Omron Sysmac Studio project IoTSampleProjectNX1P2_9 (Sysmac Studio 1.47.0.64008, StandardProject)

# Controller new_Controller_0: NX1P2-9024DT1 version 1.47
Task PrimaryTask (priority 4, period or condition 2000): MQTT_AWS, DynamoDB_AWS
Library OmronLib_MQTT_Comm_V1_0 1.0.0 (contents left out)

PROGRAM MQTT_AWS
VAR
    trigger1 : BOOL;
    ClientID : STRING[256];
    ConnectionSettings : OmronLib\MQTT_Comm\sConnectionSettings;
    Pub_Topic : STRING[512];
    Pub_PubMsg : STRING[256];
    Pub_PubSettings : OmronLib\MQTT_Comm\sPubFlags;
    Sub_Topic : STRING[512];
    ClientReference : OmronLib\MQTT_Comm\sClientReference;
    KeepAlive : UINT;
    Timeout : UINT;
    DiscardMsgTime : UINT;
    busy : BOOL;
    DiscardMsgNum : UDINT;
    SessionPresent : BOOL;
    error : BOOL;
    errorid : WORD;
    erroridex : DWORD;
    MQTTClient00 : OmronLib\MQTT_Comm\MQTTClient;
    MQTTPubString : OmronLib\MQTT_Comm\MQTTPubString;
    Pub_PacketID : UINT;
    Pub_MsgType : USINT;
    Put_Timeout : UINT;
    pub_busy : BOOL;
    pub_error : BOOL;
    pub_errorid : WORD;
    pub_erroridex : DWORD;
    MQTT : OmronLib\MQTT_Comm\MQTTSubString;
    MQTTSubString00 : OmronLib\MQTT_Comm\MQTTSubString;
    MQTTPubString00 : OmronLib\MQTT_Comm\MQTTPubString;
    Sub_RcvMsg : STRING[1986];
    Sub_SubQos : BYTE;
    Sub_Timeout : UINT;
    Sub_Status : SINT;
    Sub_Received : BOOL;
    Sub_RcvTopic : STRING[512];
    sub_error : BOOL;
    sub_errorid : WORD;
    sub_erroridex : DWORD;
    trigger2 : BOOL;
    MQTTPing00 : OmronLib\MQTT_Comm\MQTTPing;
    ping_Timeout : UINT;
    ping_busy : BOOL;
    Ping_elapsedtime : UINT;
    ping_error : BOOL;
    ping_errorid : WORD;
    ping_erroridex : DWORD;
    trigger3 : BOOL;
    trigger4 : BOOL;
    Pub_Timeout : UINT;
    trigger5 : BOOL;
    MQTTPubAry00 : OmronLib\MQTT_Comm\MQTTPubAryByte;
    Pub_MsgAry : ARRAY[0..65534] OF BYTE;
    Pub_MsgSize : UINT;
    pubary_busy : BOOL;
    pubary_error : BOOL;
    pubary_errorid : WORD;
    pubary_erroridex : DWORD;
    trigger6 : BOOL;
    MQTTSubAry00 : OmronLib\MQTT_Comm\MQTTSubAryByte;
    SubAry_RcvMsg : ARRAY[0..65534] OF BYTE;
    SubAry_SubQoS : BYTE;
    Subary_Status : SINT;
    SubAry_Received : BOOL;
    SubAry_MsgSize : UINT;
    SubAry_RcvTopic : STRING[512];
    subary_error : BOOL;
    subary_errorid : WORD;
    subary_erroridex : DWORD;
    RcvMsg : STRING[1986];
    tmpAryStr : ARRAY[0..1985] OF BYTE;
END_VAR
VAR
    _e1 : R_TRIG;
    _e2 : R_TRIG;
    _e3 : R_TRIG;
END_VAR

(* Section Section0: ladder, written here as Structured Text *)

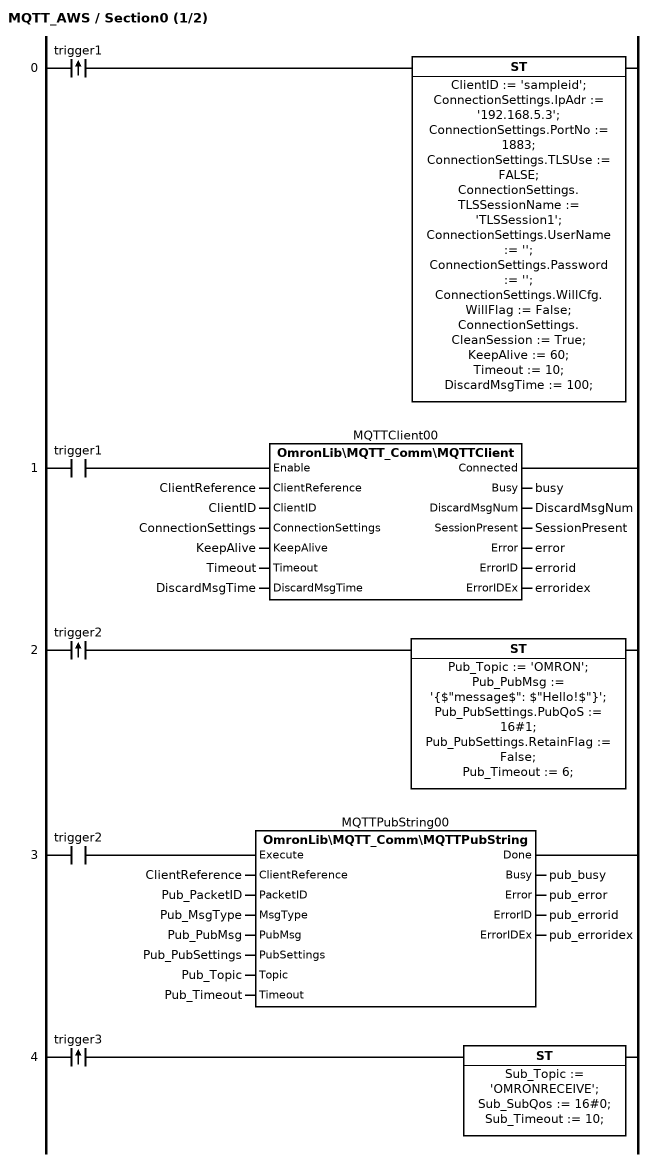
(* Rung 0 *)
_e1(CLK := trigger1);
IF _e1.Q THEN
    ClientID := 'sampleid';
    
    ConnectionSettings.IpAdr := '192.168.5.3';
    ConnectionSettings.PortNo := 1883;
    ConnectionSettings.TLSUse := FALSE;
    
    ConnectionSettings.TLSSessionName := 'TLSSession1';
    
    ConnectionSettings.UserName := '';
    ConnectionSettings.Password := '';
    ConnectionSettings.WillCfg.WillFlag := False;
    ConnectionSettings.CleanSession := True;
    
    KeepAlive := 60;
    Timeout := 10;
    DiscardMsgTime := 100;
END_IF;
(* Rung 1 *)
MQTTClient00(Enable := trigger1, ClientReference := ClientReference, ClientID := ClientID, ConnectionSettings := ConnectionSettings, KeepAlive := KeepAlive, Timeout := Timeout, DiscardMsgTime := DiscardMsgTime, Busy => busy, DiscardMsgNum => DiscardMsgNum, SessionPresent => SessionPresent, Error => error, ErrorID => errorid, ErrorIDEx => erroridex);
(* Rung 2 *)
_e2(CLK := trigger2);
IF _e2.Q THEN
    Pub_Topic := 'OMRON';
    
    Pub_PubMsg := '{$"message$": $"Hello!$"}';
    Pub_PubSettings.PubQoS := 16#1;
    Pub_PubSettings.RetainFlag := False;
    
    Pub_Timeout := 6;
END_IF;
(* Rung 3 *)
MQTTPubString00(Execute := trigger2, ClientReference := ClientReference, PacketID := Pub_PacketID, MsgType := Pub_MsgType, PubMsg := Pub_PubMsg, PubSettings := Pub_PubSettings, Topic := Pub_Topic, Timeout := Pub_Timeout, Busy => pub_busy, Error => pub_error, ErrorID => pub_errorid, ErrorIDEx => pub_erroridex);
(* Rung 4 *)
_e3(CLK := trigger3);
IF _e3.Q THEN
    Sub_Topic := 'OMRONRECEIVE';
    
    Sub_SubQos := 16#0;
    Sub_Timeout := 10;
END_IF;

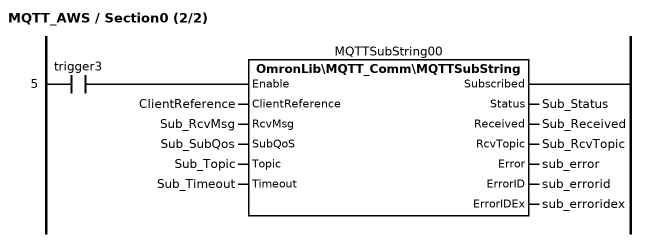
(* Rung 5 *)
MQTTSubString00(Enable := trigger3, ClientReference := ClientReference, RcvMsg := Sub_RcvMsg, SubQoS := Sub_SubQos, Topic := Sub_Topic, Timeout := Sub_Timeout, Status => Sub_Status, Received => Sub_Received, RcvTopic => Sub_RcvTopic, Error => sub_error, ErrorID => sub_errorid, ErrorIDEx => sub_erroridex);
END_PROGRAM

PROGRAM DynamoDB_AWS
VAR
    trigger1 : BOOL;
    ClientID : STRING[256];
    ConnectionSettings : OmronLib\MQTT_Comm\sConnectionSettings;
    Pub_Topic : STRING[512];
    Pub_PubMsg : STRING[256];
    Pub_PubSettings : OmronLib\MQTT_Comm\sPubFlags;
    Sub_Topic : STRING[512];
    ClientReference : OmronLib\MQTT_Comm\sClientReference;
    KeepAlive : UINT;
    Timeout : UINT;
    DiscardMsgTime : UINT;
    busy : BOOL;
    DiscardMsgNum : UDINT;
    SessionPresent : BOOL;
    error : BOOL;
    errorid : WORD;
    erroridex : DWORD;
    MQTTClient00 : OmronLib\MQTT_Comm\MQTTClient;
    MQTTPubString : OmronLib\MQTT_Comm\MQTTPubString;
    Pub_PacketID : UINT;
    Pub_MsgType : USINT;
    Put_Timeout : UINT;
    pub_busy : BOOL;
    pub_error : BOOL;
    pub_errorid : WORD;
    pub_erroridex : DWORD;
    MQTT : OmronLib\MQTT_Comm\MQTTSubString;
    MQTTSubString00 : OmronLib\MQTT_Comm\MQTTSubString;
    MQTTPubString00 : OmronLib\MQTT_Comm\MQTTPubString;
    Sub_RcvMsg : STRING[1986];
    Sub_SubQos : BYTE;
    Sub_Timeout : UINT;
    Sub_Status : SINT;
    Sub_Received : BOOL;
    Sub_RcvTopic : STRING[512];
    sub_error : BOOL;
    sub_errorid : WORD;
    sub_erroridex : DWORD;
    trigger2 : BOOL;
    MQTTPing00 : OmronLib\MQTT_Comm\MQTTPing;
    ping_Timeout : UINT;
    ping_busy : BOOL;
    Ping_elapsedtime : UINT;
    ping_error : BOOL;
    ping_errorid : WORD;
    ping_erroridex : DWORD;
    trigger3 : BOOL;
    trigger4 : BOOL;
    Pub_Timeout : UINT;
    trigger5 : BOOL;
    MQTTPubAry00 : OmronLib\MQTT_Comm\MQTTPubAryByte;
    Pub_MsgAry : ARRAY[0..65534] OF BYTE;
    Pub_MsgSize : UINT;
    pubary_busy : BOOL;
    pubary_error : BOOL;
    pubary_errorid : WORD;
    pubary_erroridex : DWORD;
    trigger6 : BOOL;
    MQTTSubAry00 : OmronLib\MQTT_Comm\MQTTSubAryByte;
    SubAry_RcvMsg : ARRAY[0..65534] OF BYTE;
    SubAry_SubQoS : BYTE;
    Subary_Status : SINT;
    SubAry_Received : BOOL;
    SubAry_MsgSize : UINT;
    SubAry_RcvTopic : STRING[512];
    subary_error : BOOL;
    subary_errorid : WORD;
    subary_erroridex : DWORD;
    RcvMsg : STRING[1986];
    tmpAryStr : ARRAY[0..1985] OF BYTE;
END_VAR
VAR
    _e1 : R_TRIG;
    _e2 : R_TRIG;
END_VAR

(* Section Section0: ladder, written here as Structured Text *)

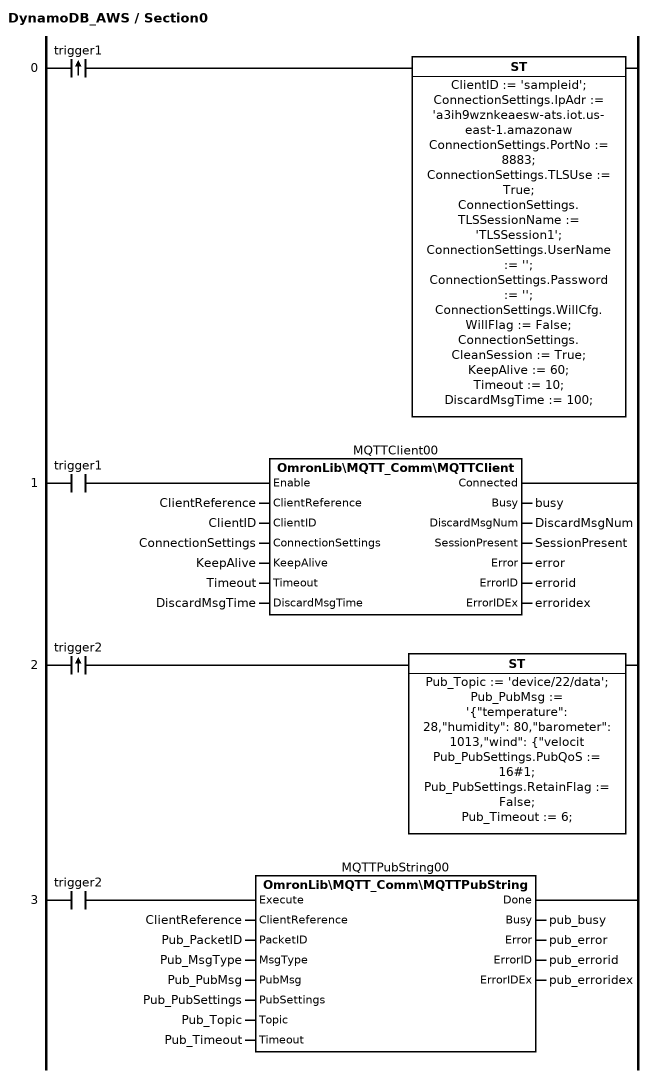
(* Rung 0 *)
_e1(CLK := trigger1);
IF _e1.Q THEN
    ClientID := 'sampleid';
    
    ConnectionSettings.IpAdr := 'a3ih9wznkeaesw-ats.iot.us-east-1.amazonaws.com';
    ConnectionSettings.PortNo := 8883;
    ConnectionSettings.TLSUse := True;
    
    ConnectionSettings.TLSSessionName := 'TLSSession1';
    
    ConnectionSettings.UserName := '';
    ConnectionSettings.Password := '';
    ConnectionSettings.WillCfg.WillFlag := False;
    ConnectionSettings.CleanSession := True;
    
    KeepAlive := 60;
    Timeout := 10;
    DiscardMsgTime := 100;
END_IF;
(* Rung 1 *)
MQTTClient00(Enable := trigger1, ClientReference := ClientReference, ClientID := ClientID, ConnectionSettings := ConnectionSettings, KeepAlive := KeepAlive, Timeout := Timeout, DiscardMsgTime := DiscardMsgTime, Busy => busy, DiscardMsgNum => DiscardMsgNum, SessionPresent => SessionPresent, Error => error, ErrorID => errorid, ErrorIDEx => erroridex);
(* Rung 2 *)
_e2(CLK := trigger2);
IF _e2.Q THEN
    Pub_Topic := 'device/22/data';
    
    Pub_PubMsg := 
    '{"temperature": 28,"humidity": 80,"barometer": 1013,"wind": {"velocity": 22,"bearing": 255}}';
    
    Pub_PubSettings.PubQoS := 16#1;
    Pub_PubSettings.RetainFlag := False;
    
    Pub_Timeout := 6;
END_IF;
(* Rung 3 *)
MQTTPubString00(Execute := trigger2, ClientReference := ClientReference, PacketID := Pub_PacketID, MsgType := Pub_MsgType, PubMsg := Pub_PubMsg, PubSettings := Pub_PubSettings, Topic := Pub_Topic, Timeout := Pub_Timeout, Busy => pub_busy, Error => pub_error, ErrorID => pub_errorid, ErrorIDEx => pub_erroridex);
END_PROGRAM